PROGRAM MAIN
VAR
	iHeartbeat : ULINT;
	
	st_comm : ST_PyADS;
END_VAR

iHeartbeat := iHeartbeat + 1;

END_PROGRAM

(* stored: Version 1.1.0.1, ProductVersion 3.1.4024.12
   POU MAIN: Id {df0e651f-fc01-4c13-90cd-d475f9fa8ba2}, SpecialFunc None *)
